// TwinCAT 3 PLC project plc_tmo_test_vac
// ProgramVersion: 3.1.4022.7
// libraries:
//   LCLS General, * (SLAC)
//   LCLS Vacuum, * (SLAC - LCLS)
//   LCLSVacuumSerialDriverLib, * (SLAC - LCLS)
//   Tc2_SerialCom, * (Beckhoff Automation GmbH)
//   Tc2_Standard, * (Beckhoff Automation GmbH)
//   Tc2_System, * (Beckhoff Automation GmbH)
//   Tc3_Module, * (Beckhoff Automation GmbH)
// project tree:
//   GVLs/ GVL_COM.TcGVL, GVL_Devices.TcGVL
//   / PlcTask.TcTTO
//   POUs/ MAIN.TcPOU, PRG_COM.TcPOU
// real-time tasks:
//   TASK PlcTask: cycle T#10ms, priority 20, ADS port 350
// motion (NC):
// I/O:
//   DEVICE Device 1 (EtherCAT), AmsNetId 172.21.148.66.2.1
//     Term 1 (EK1200) [EK1200-5000 EtherCAT Power supply (2A E-Bus)]
//       Term 2 (EL7041) [EL7041 1Ch. Stepper motor output stage (50V, 5A)]
//       Term 3 (EL6692) [EL6692 EtherCAT Bridge terminal (Primary)]
//       Term 4 (EK1110) [EK1110 EtherCAT extension]
//     LAMP_CLSTR1_PNL1_EP01_EP2338-0002 [EP2338-0002 8 Ch. Dig. Input/Output 24V, 0,5A, M12]
//     LAMP_CLSTR1_PNL1_EP02_EP2624-0002 [EP2624-0002 4Ch. Relay Output, NO (125V AC / 30V DC)]
//     LAMP_CLSTR1_PNL1_EP03_EP6002-0002 [EP6002-0002 Interface (RS232/422/485)]
// variable links:
//   plc_tmo_test_vac Instance <-> Device 1 (EtherCAT)/LAMP_CLSTR1_PNL1_EP01_EP2338-0002
//     PlcTask Inputs/GVL_Devices.LAMP_CLSTR1_PTM_01.i_xAtSpd <-> Channel 1/Input
//     PlcTask Inputs/GVL_Devices.LAMP_CLSTR1_PTM_01.i_xFaultNC <-> Channel 2/Input
//     PlcTask Inputs/GVL_Devices.LAMP_CLSTR1_PTM_01.i_xRemote <-> Channel 3/Input
//   plc_tmo_test_vac Instance <-> Device 1 (EtherCAT)/LAMP_CLSTR1_PNL1_EP02_EP2624-0002
//     PlcTask Outputs/GVL_Devices.LAMP_CLSTR1_PTM_01.q_RunDO <-> Channel 1/Output
//     PlcTask Outputs/GVL_Devices.LAMP_CLSTR1_PTM_01.q_xReset <-> Channel 2/Output
//   plc_tmo_test_vac Instance <-> Device 1 (EtherCAT)/LAMP_CLSTR1_PNL1_EP03_EP6002-0002
//     PlcTask Inputs/GVL_COM.stComIn_LAMP_CLSTR1_PTM_01/D[0] <-> COM TxPDO-Map Inputs Channel 1/Data In 0
//     PlcTask Inputs/GVL_COM.stComIn_LAMP_CLSTR1_PTM_01/D[10] <-> COM TxPDO-Map Inputs Channel 1/Data In 10
//     PlcTask Inputs/GVL_COM.stComIn_LAMP_CLSTR1_PTM_01/D[11] <-> COM TxPDO-Map Inputs Channel 1/Data In 11
//     PlcTask Inputs/GVL_COM.stComIn_LAMP_CLSTR1_PTM_01/D[12] <-> COM TxPDO-Map Inputs Channel 1/Data In 12
//     PlcTask Inputs/GVL_COM.stComIn_LAMP_CLSTR1_PTM_01/D[13] <-> COM TxPDO-Map Inputs Channel 1/Data In 13
//     PlcTask Inputs/GVL_COM.stComIn_LAMP_CLSTR1_PTM_01/D[14] <-> COM TxPDO-Map Inputs Channel 1/Data In 14
//     PlcTask Inputs/GVL_COM.stComIn_LAMP_CLSTR1_PTM_01/D[15] <-> COM TxPDO-Map Inputs Channel 1/Data In 15
//     PlcTask Inputs/GVL_COM.stComIn_LAMP_CLSTR1_PTM_01/D[16] <-> COM TxPDO-Map Inputs Channel 1/Data In 16
//     PlcTask Inputs/GVL_COM.stComIn_LAMP_CLSTR1_PTM_01/D[17] <-> COM TxPDO-Map Inputs Channel 1/Data In 17
//     PlcTask Inputs/GVL_COM.stComIn_LAMP_CLSTR1_PTM_01/D[18] <-> COM TxPDO-Map Inputs Channel 1/Data In 18
//     PlcTask Inputs/GVL_COM.stComIn_LAMP_CLSTR1_PTM_01/D[19] <-> COM TxPDO-Map Inputs Channel 1/Data In 19
//     PlcTask Inputs/GVL_COM.stComIn_LAMP_CLSTR1_PTM_01/D[1] <-> COM TxPDO-Map Inputs Channel 1/Data In 1
//     PlcTask Inputs/GVL_COM.stComIn_LAMP_CLSTR1_PTM_01/D[20] <-> COM TxPDO-Map Inputs Channel 1/Data In 20
//     PlcTask Inputs/GVL_COM.stComIn_LAMP_CLSTR1_PTM_01/D[21] <-> COM TxPDO-Map Inputs Channel 1/Data In 21
//     PlcTask Inputs/GVL_COM.stComIn_LAMP_CLSTR1_PTM_01/D[2] <-> COM TxPDO-Map Inputs Channel 1/Data In 2
//     PlcTask Inputs/GVL_COM.stComIn_LAMP_CLSTR1_PTM_01/D[3] <-> COM TxPDO-Map Inputs Channel 1/Data In 3
//     PlcTask Inputs/GVL_COM.stComIn_LAMP_CLSTR1_PTM_01/D[4] <-> COM TxPDO-Map Inputs Channel 1/Data In 4
//     PlcTask Inputs/GVL_COM.stComIn_LAMP_CLSTR1_PTM_01/D[5] <-> COM TxPDO-Map Inputs Channel 1/Data In 5
//     PlcTask Inputs/GVL_COM.stComIn_LAMP_CLSTR1_PTM_01/D[6] <-> COM TxPDO-Map Inputs Channel 1/Data In 6
//     PlcTask Inputs/GVL_COM.stComIn_LAMP_CLSTR1_PTM_01/D[7] <-> COM TxPDO-Map Inputs Channel 1/Data In 7
//     PlcTask Inputs/GVL_COM.stComIn_LAMP_CLSTR1_PTM_01/D[8] <-> COM TxPDO-Map Inputs Channel 1/Data In 8
//     PlcTask Inputs/GVL_COM.stComIn_LAMP_CLSTR1_PTM_01/D[9] <-> COM TxPDO-Map Inputs Channel 1/Data In 9
//     PlcTask Inputs/GVL_COM.stComIn_LAMP_CLSTR1_PTM_01/Status <-> COM TxPDO-Map Inputs Channel 1/Status
//     PlcTask Outputs/GVL_COM.stComOut_LAMP_CLSTR1_PTM_01/Ctrl <-> COM RxPDO-Map Outputs Channel 1/Ctrl
//     PlcTask Outputs/GVL_COM.stComOut_LAMP_CLSTR1_PTM_01/D[0] <-> COM RxPDO-Map Outputs Channel 1/Data Out 0
//     PlcTask Outputs/GVL_COM.stComOut_LAMP_CLSTR1_PTM_01/D[10] <-> COM RxPDO-Map Outputs Channel 1/Data Out 10
//     PlcTask Outputs/GVL_COM.stComOut_LAMP_CLSTR1_PTM_01/D[11] <-> COM RxPDO-Map Outputs Channel 1/Data Out 11
//     PlcTask Outputs/GVL_COM.stComOut_LAMP_CLSTR1_PTM_01/D[12] <-> COM RxPDO-Map Outputs Channel 1/Data Out 12
//     PlcTask Outputs/GVL_COM.stComOut_LAMP_CLSTR1_PTM_01/D[13] <-> COM RxPDO-Map Outputs Channel 1/Data Out 13
//     PlcTask Outputs/GVL_COM.stComOut_LAMP_CLSTR1_PTM_01/D[14] <-> COM RxPDO-Map Outputs Channel 1/Data Out 14
//     PlcTask Outputs/GVL_COM.stComOut_LAMP_CLSTR1_PTM_01/D[15] <-> COM RxPDO-Map Outputs Channel 1/Data Out 15
//     PlcTask Outputs/GVL_COM.stComOut_LAMP_CLSTR1_PTM_01/D[16] <-> COM RxPDO-Map Outputs Channel 1/Data Out 16
//     PlcTask Outputs/GVL_COM.stComOut_LAMP_CLSTR1_PTM_01/D[17] <-> COM RxPDO-Map Outputs Channel 1/Data Out 17
//     PlcTask Outputs/GVL_COM.stComOut_LAMP_CLSTR1_PTM_01/D[18] <-> COM RxPDO-Map Outputs Channel 1/Data Out 18
//     PlcTask Outputs/GVL_COM.stComOut_LAMP_CLSTR1_PTM_01/D[19] <-> COM RxPDO-Map Outputs Channel 1/Data Out 19
//     PlcTask Outputs/GVL_COM.stComOut_LAMP_CLSTR1_PTM_01/D[1] <-> COM RxPDO-Map Outputs Channel 1/Data Out 1
//     PlcTask Outputs/GVL_COM.stComOut_LAMP_CLSTR1_PTM_01/D[20] <-> COM RxPDO-Map Outputs Channel 1/Data Out 20
//     PlcTask Outputs/GVL_COM.stComOut_LAMP_CLSTR1_PTM_01/D[21] <-> COM RxPDO-Map Outputs Channel 1/Data Out 21
//     PlcTask Outputs/GVL_COM.stComOut_LAMP_CLSTR1_PTM_01/D[2] <-> COM RxPDO-Map Outputs Channel 1/Data Out 2
//     PlcTask Outputs/GVL_COM.stComOut_LAMP_CLSTR1_PTM_01/D[3] <-> COM RxPDO-Map Outputs Channel 1/Data Out 3
//     PlcTask Outputs/GVL_COM.stComOut_LAMP_CLSTR1_PTM_01/D[4] <-> COM RxPDO-Map Outputs Channel 1/Data Out 4
//     PlcTask Outputs/GVL_COM.stComOut_LAMP_CLSTR1_PTM_01/D[5] <-> COM RxPDO-Map Outputs Channel 1/Data Out 5
//     PlcTask Outputs/GVL_COM.stComOut_LAMP_CLSTR1_PTM_01/D[6] <-> COM RxPDO-Map Outputs Channel 1/Data Out 6
//     PlcTask Outputs/GVL_COM.stComOut_LAMP_CLSTR1_PTM_01/D[7] <-> COM RxPDO-Map Outputs Channel 1/Data Out 7
//     PlcTask Outputs/GVL_COM.stComOut_LAMP_CLSTR1_PTM_01/D[8] <-> COM RxPDO-Map Outputs Channel 1/Data Out 8
//     PlcTask Outputs/GVL_COM.stComOut_LAMP_CLSTR1_PTM_01/D[9] <-> COM RxPDO-Map Outputs Channel 1/Data Out 9

CONFIGURATION plc_tmo_test_vac
    RESOURCE PLC ON TwinCAT3
        TASK PlcTask(INTERVAL := T#10ms, PRIORITY := 20);
        PROGRAM MAIN WITH PlcTask : MAIN;
    END_RESOURCE
END_CONFIGURATION

// ---- GVLs/GVL_COM.TcGVL
{attribute 'qualified_only'}
VAR_GLOBAL
	
// Define COM Ports/Buffers incl. library Tc2_SerialCom
SerialRXBuffer_LAMP_CLSTR1_PTM_01 : ComBuffer;
SerialTXBuffer_LAMP_CLSTR1_PTM_01 : ComBuffer;

// Serial Terminal
fbSerialLineControl_LAMP_CLSTR1_PTM_01: SerialLineControl;

//SERIAL IO
	{attribute	'TcLinkTo'	:=	'.Status:=TIIB[LAMP_CLSTR1_PNL1_EP03_EP6002-0002]^COM TxPDO-Map Inputs Channel 1^Status;
								 .D[0]:=TIIB[LAMP_CLSTR1_PNL1_EP03_EP6002-0002]^COM TxPDO-Map Inputs Channel 1^Data In 0;
								 .D[1]:=TIIB[LAMP_CLSTR1_PNL1_EP03_EP6002-0002]^COM TxPDO-Map Inputs Channel 1^Data In 1;
								 .D[2]:=TIIB[LAMP_CLSTR1_PNL1_EP03_EP6002-0002]^COM TxPDO-Map Inputs Channel 1^Data In 2;
								 .D[3]:=TIIB[LAMP_CLSTR1_PNL1_EP03_EP6002-0002]^COM TxPDO-Map Inputs Channel 1^Data In 3;
								 .D[4]:=TIIB[LAMP_CLSTR1_PNL1_EP03_EP6002-0002]^COM TxPDO-Map Inputs Channel 1^Data In 4;
								 .D[5]:=TIIB[LAMP_CLSTR1_PNL1_EP03_EP6002-0002]^COM TxPDO-Map Inputs Channel 1^Data In 5;
								 .D[6]:=TIIB[LAMP_CLSTR1_PNL1_EP03_EP6002-0002]^COM TxPDO-Map Inputs Channel 1^Data In 6;
								 .D[7]:=TIIB[LAMP_CLSTR1_PNL1_EP03_EP6002-0002]^COM TxPDO-Map Inputs Channel 1^Data In 7;
								 .D[8]:=TIIB[LAMP_CLSTR1_PNL1_EP03_EP6002-0002]^COM TxPDO-Map Inputs Channel 1^Data In 8;
								 .D[9]:=TIIB[LAMP_CLSTR1_PNL1_EP03_EP6002-0002]^COM TxPDO-Map Inputs Channel 1^Data In 9;
								 .D[10]:=TIIB[LAMP_CLSTR1_PNL1_EP03_EP6002-0002]^COM TxPDO-Map Inputs Channel 1^Data In 10;
								 .D[11]:=TIIB[LAMP_CLSTR1_PNL1_EP03_EP6002-0002]^COM TxPDO-Map Inputs Channel 1^Data In 11;
								 .D[12]:=TIIB[LAMP_CLSTR1_PNL1_EP03_EP6002-0002]^COM TxPDO-Map Inputs Channel 1^Data In 12;
								 .D[13]:=TIIB[LAMP_CLSTR1_PNL1_EP03_EP6002-0002]^COM TxPDO-Map Inputs Channel 1^Data In 13;
								 .D[14]:=TIIB[LAMP_CLSTR1_PNL1_EP03_EP6002-0002]^COM TxPDO-Map Inputs Channel 1^Data In 14;
								 .D[15]:=TIIB[LAMP_CLSTR1_PNL1_EP03_EP6002-0002]^COM TxPDO-Map Inputs Channel 1^Data In 15;
								 .D[16]:=TIIB[LAMP_CLSTR1_PNL1_EP03_EP6002-0002]^COM TxPDO-Map Inputs Channel 1^Data In 16;
								 .D[17]:=TIIB[LAMP_CLSTR1_PNL1_EP03_EP6002-0002]^COM TxPDO-Map Inputs Channel 1^Data In 17;
								 .D[18]:=TIIB[LAMP_CLSTR1_PNL1_EP03_EP6002-0002]^COM TxPDO-Map Inputs Channel 1^Data In 18;
								 .D[19]:=TIIB[LAMP_CLSTR1_PNL1_EP03_EP6002-0002]^COM TxPDO-Map Inputs Channel 1^Data In 19;
								 .D[20]:=TIIB[LAMP_CLSTR1_PNL1_EP03_EP6002-0002]^COM TxPDO-Map Inputs Channel 1^Data In 20;
								 .D[21]:=TIIB[LAMP_CLSTR1_PNL1_EP03_EP6002-0002]^COM TxPDO-Map Inputs Channel 1^Data In 21;
	'}
	stComIn_LAMP_CLSTR1_PTM_01		AT %I*	:	EL6inData22B;
	
	{attribute	'TcLinkTo'	:=	'.Ctrl:=TIIB[LAMP_CLSTR1_PNL1_EP03_EP6002-0002]^COM RxPDO-Map Outputs Channel 1^Ctrl;
								 .D[0]:=TIIB[LAMP_CLSTR1_PNL1_EP03_EP6002-0002]^COM RxPDO-Map Outputs Channel 1^Data Out 0;
								 .D[1]:=TIIB[LAMP_CLSTR1_PNL1_EP03_EP6002-0002]^COM RxPDO-Map Outputs Channel 1^Data Out 1;
								 .D[2]:=TIIB[LAMP_CLSTR1_PNL1_EP03_EP6002-0002]^COM RxPDO-Map Outputs Channel 1^Data Out 2;
								 .D[3]:=TIIB[LAMP_CLSTR1_PNL1_EP03_EP6002-0002]^COM RxPDO-Map Outputs Channel 1^Data Out 3;
								 .D[4]:=TIIB[LAMP_CLSTR1_PNL1_EP03_EP6002-0002]^COM RxPDO-Map Outputs Channel 1^Data Out 4;
								 .D[5]:=TIIB[LAMP_CLSTR1_PNL1_EP03_EP6002-0002]^COM RxPDO-Map Outputs Channel 1^Data Out 5;
								 .D[6]:=TIIB[LAMP_CLSTR1_PNL1_EP03_EP6002-0002]^COM RxPDO-Map Outputs Channel 1^Data Out 6;
								 .D[7]:=TIIB[LAMP_CLSTR1_PNL1_EP03_EP6002-0002]^COM RxPDO-Map Outputs Channel 1^Data Out 7;
								 .D[8]:=TIIB[LAMP_CLSTR1_PNL1_EP03_EP6002-0002]^COM RxPDO-Map Outputs Channel 1^Data Out 8;
								 .D[9]:=TIIB[LAMP_CLSTR1_PNL1_EP03_EP6002-0002]^COM RxPDO-Map Outputs Channel 1^Data Out 9;
								 .D[10]:=TIIB[LAMP_CLSTR1_PNL1_EP03_EP6002-0002]^COM RxPDO-Map Outputs Channel 1^Data Out 10;
								 .D[11]:=TIIB[LAMP_CLSTR1_PNL1_EP03_EP6002-0002]^COM RxPDO-Map Outputs Channel 1^Data Out 11;
								 .D[12]:=TIIB[LAMP_CLSTR1_PNL1_EP03_EP6002-0002]^COM RxPDO-Map Outputs Channel 1^Data Out 12;
								 .D[13]:=TIIB[LAMP_CLSTR1_PNL1_EP03_EP6002-0002]^COM RxPDO-Map Outputs Channel 1^Data Out 13;
								 .D[14]:=TIIB[LAMP_CLSTR1_PNL1_EP03_EP6002-0002]^COM RxPDO-Map Outputs Channel 1^Data Out 14;
								 .D[15]:=TIIB[LAMP_CLSTR1_PNL1_EP03_EP6002-0002]^COM RxPDO-Map Outputs Channel 1^Data Out 15;
								 .D[16]:=TIIB[LAMP_CLSTR1_PNL1_EP03_EP6002-0002]^COM RxPDO-Map Outputs Channel 1^Data Out 16;
								 .D[17]:=TIIB[LAMP_CLSTR1_PNL1_EP03_EP6002-0002]^COM RxPDO-Map Outputs Channel 1^Data Out 17;
								 .D[18]:=TIIB[LAMP_CLSTR1_PNL1_EP03_EP6002-0002]^COM RxPDO-Map Outputs Channel 1^Data Out 18;
								 .D[19]:=TIIB[LAMP_CLSTR1_PNL1_EP03_EP6002-0002]^COM RxPDO-Map Outputs Channel 1^Data Out 19;
								 .D[20]:=TIIB[LAMP_CLSTR1_PNL1_EP03_EP6002-0002]^COM RxPDO-Map Outputs Channel 1^Data Out 20;
								 .D[21]:=TIIB[LAMP_CLSTR1_PNL1_EP03_EP6002-0002]^COM RxPDO-Map Outputs Channel 1^Data Out 21;
	'}
	stComOut_LAMP_CLSTR1_PTM_01		AT %Q*	:	EL6outData22B;

END_VAR

// ---- GVLs/GVL_Devices.TcGVL
{attribute 'qualified_only'}
VAR_GLOBAL
	
(*LAMP CLSTR1 Turbo Pump*)
	{attribute 'TcLinkTo' := 	'.i_xAtSpd			:=	TIIB[LAMP_CLSTR1_PNL1_EP01_EP2338-0002]^Channel 1^Input;
								 .i_xFaultNC		:=	TIIB[LAMP_CLSTR1_PNL1_EP01_EP2338-0002]^Channel 2^Input;
								 .i_xRemote			:=	TIIB[LAMP_CLSTR1_PNL1_EP01_EP2338-0002]^Channel 3^Input;
								 .q_RunDO			:=	TIIB[LAMP_CLSTR1_PNL1_EP02_EP2624-0002]^Channel 1^Output;
								 .q_xReset 			:=	TIIB[LAMP_CLSTR1_PNL1_EP02_EP2624-0002]^Channel 2^Output				 
	'}
	{attribute 'pytmc' := '
		pv: LAMP:CLSTR1:PTM:01
		io: io
	'}
	LAMP_CLSTR1_PTM_01 : FB_PTM_Pfeiffer;

(*Pfeiffer*)
	// They share the same serial port
	st_Pfeiffer_CTRL_LAMP_CLSTR1_PTM_01 		: ARRAY[1..20] OF ST_PfeifferControl;
	st_Pfeiffer_RBK_LAMP_CLSTR1_PTM_01 			: ARRAY[1..20] OF ST_PfeifferStatus;
	fb_PfeifferCom_LAMP_CLSTR1_PTM_01 			: FB_PFEIFFER_COM;
	
END_VAR

// ---- POUs/MAIN.TcPOU
PROGRAM MAIN
VAR	
	LAMP_CLSTR1_PTM_01: FB_PTM_Pfeiffer;
	st_Pfeiffer_CTRL_LAMP_CLSTR1_PTM_01: ST_PfeifferControl;
	xEnableComm: INT;
	fb_PfeifferCom_LAMP_CLSTR1_PTM_01: FB_PFEIFFER_COM;
END_VAR

(*TURBO Pump*)
LAMP_CLSTR1_PTM_01(i_xExtIlkOK:= True, iq_stPTM=> );

(*Serial Communication*)
(*Assign adresses to the pfeiffer controllers connected to this serial terminal*)
st_Pfeiffer_CTRL_LAMP_CLSTR1_PTM_01.iSerialAddress :=1;
st_Pfeiffer_CTRL_LAMP_CLSTR1_PTM_01.xEnableComm := TRUE;

(* Instanitate the Function block for serial communication with Pfeiffer*)
	
fb_PfeifferCom_LAMP_CLSTR1_PTM_01(astPfeifferControl := st_Pfeiffer_CTRL_LAMP_CLSTR1_PTM_01,
			   				  astPfeifferStatus:= st_Pfeiffer_RBK_LAMP_CLSTR1_PTM_01,
							  SerialRXBuffer:= SerialRXBuffer_LAMP_CLSTR1_PTM_01,
							  SerialTXBuffer:= SerialTXBuffer_LAMP_CLSTR1_PTM_01);


(* Copy Status Pv's into the PTM structure*)
LAMP_CLSTR1_PTM_01.M_Serial_IO(st_Pfeiffer_RBK:= st_Pfeiffer_RBK_LAMP_CLSTR1_PTM_01[1], st_Pfeiffer_CTRL:= st_Pfeiffer_CTRL_LAMP_CLSTR1_PTM_01[1]);

END_PROGRAM

// ---- POUs/PRG_COM.TcPOU
PROGRAM PRG_COM
VAR
END_VAR

(*Instanitate Serial port com function *) 
fbSerialLineControl_LAMP_CLSTR1_PTM_01(
	Mode:= SERIALLINEMODE_EL6_22B,
	pComIn:= ADR(stComIn_LAMP_CLSTR1_PTM_01),
	pComOut:=ADR(stComOut_LAMP_CLSTR1_PTM_01),
	SizeComIn:= SIZEOF(stComIn_LAMP_CLSTR1_PTM_01),
	TxBuffer:= SerialTXBuffer_LAMP_CLSTR1_PTM_01,
	RxBuffer:= SerialRXBuffer_LAMP_CLSTR1_PTM_01,
	Error=> ,
	ErrorID=> );

END_PROGRAM
